SUBAPPLICATION Uebung_006a3_AX (* SR und T-Flip-Flop mit 3x IE; links/rechtslauf *)
  (* Standard: 61499-2; Description: Copyright (c) 2023 Meisterschulen am Ostbahnhof This program and the accompanying materials are made available under the terms of the Eclipse Public License 2.0 which is available at https://www.eclipse.org/legal/epl-2.0/ SPDX-License-Identifier: EPL-2.0 *)
  (* Version 1.0, 2023-10-23, Franz Höpfinger, Meisterschulen am Ostbahnhof, initial API and implementation and/or initial documentation *)
  PACKAGE Uebungen;
  IMPORT logiBUS::io::DI::logiBUS_DI::Input_I1;
  IMPORT logiBUS::io::DI::logiBUS_DI::Input_I2;
  IMPORT logiBUS::io::DI::logiBUS_DI::Input_I3;
  IMPORT logiBUS::io::DI::logiBUS_DI_Events::BUTTON_SINGLE_CLICK;
  IMPORT logiBUS::io::DQ::logiBUS_DO::Output_Q1;
  IMPORT logiBUS::io::DQ::logiBUS_DO::Output_Q2;
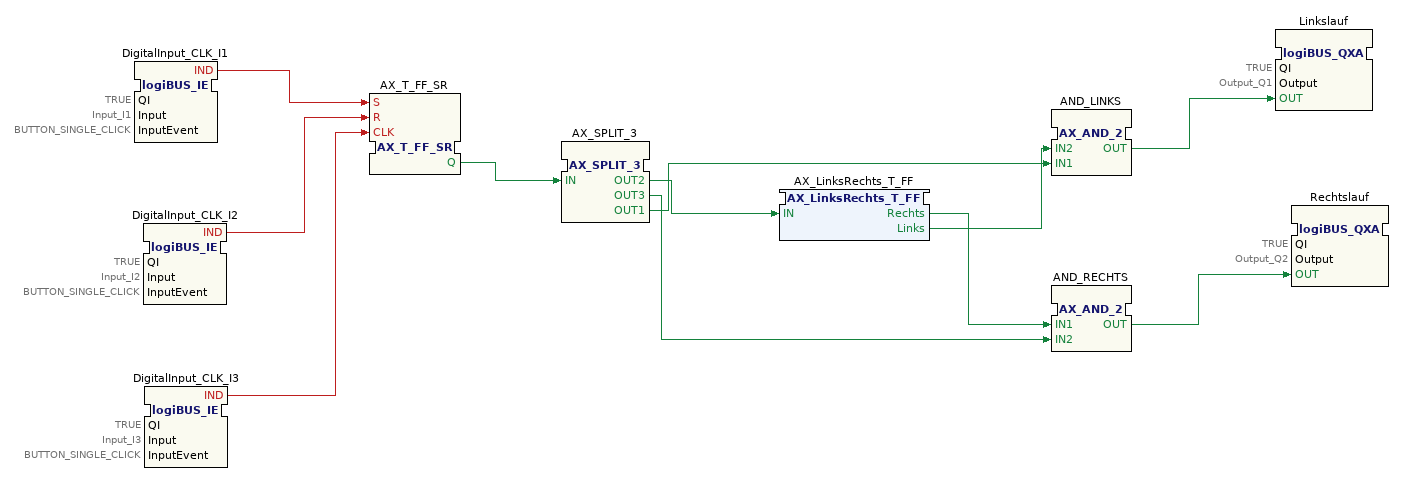
  FBS
    DigitalInput_CLK_I1 : logiBUS::io::DI::logiBUS_IE(QI := TRUE, Input := Input_I1, InputEvent := BUTTON_SINGLE_CLICK);
    DigitalInput_CLK_I2 : logiBUS::io::DI::logiBUS_IE(QI := TRUE, Input := Input_I2, InputEvent := BUTTON_SINGLE_CLICK);
    AX_T_FF_SR : adapter::events::unidirectional::AX_T_FF_SR;
    DigitalInput_CLK_I3 : logiBUS::io::DI::logiBUS_IE(QI := TRUE, Input := Input_I3, InputEvent := BUTTON_SINGLE_CLICK);
    AND_LINKS : adapter::booleanOperators::AX_AND_2;
    Rechtslauf : logiBUS::io::DQ::logiBUS_QXA(QI := TRUE, Output := Output_Q2);
    Linkslauf : logiBUS::io::DQ::logiBUS_QXA(QI := TRUE, Output := Output_Q1);
    AND_RECHTS : adapter::booleanOperators::AX_AND_2;
    AX_SPLIT_3 : adapter::events::unidirectional::AX_SPLIT_3;
  END_FBS
  SUBAPPS
    AX_LinksRechts_T_FF : MyLib::sys::AX_LinksRechts_T_FF;
  END_SUBAPPS
  EVENT_CONNECTIONS
    DigitalInput_CLK_I1.IND TO AX_T_FF_SR.S;
    DigitalInput_CLK_I2.IND TO AX_T_FF_SR.R;
    DigitalInput_CLK_I3.IND TO AX_T_FF_SR.CLK;
  END_CONNECTIONS
  ADAPTER_CONNECTIONS
    AND_RECHTS.OUT TO Rechtslauf.OUT;
    AND_LINKS.OUT TO Linkslauf.OUT;
    AX_LinksRechts_T_FF.Rechts TO AND_RECHTS.IN1;
    AX_LinksRechts_T_FF.Links TO AND_LINKS.IN2;
    AX_T_FF_SR.Q TO AX_SPLIT_3.IN;
    AX_SPLIT_3.OUT2 TO AX_LinksRechts_T_FF.IN;
    AX_SPLIT_3.OUT3 TO AND_RECHTS.IN2;
    AX_SPLIT_3.OUT1 TO AND_LINKS.IN1;
  END_CONNECTIONS
END_SUBAPPLICATION
